// SIMATIC S7-200 project (STEP 7-Micro/WIN), CPU 224 REL 02.01

SYMBOL_TABLE USUARIO1
P_MARCHA         I0.0
P_PARO           I0.1
P_DESACTIVACION  I0.2
FCEL1            I0.3
FCEL2            I0.4
F_C_F_LINEA      I0.5
S_PRESION        I0.6
F_C_T2           I0.7
F_C_T3           I1.0
CT_M_1           Q0.0
CT_M_2           Q0.1
CT_M_3           Q0.2
P_DESPLA_P       Q0.3
P_ELEVACION      Q0.4
P_BAJADA         Q0.5
P_T3             Q0.6
MEM_CP           M10.1
MEM_CG           M10.3
PT_2             Q0.7
END_SYMBOL_TABLE

ORGANIZATION_BLOCK PRINCIPAL:OB1
TITLE=COMENTARIOS DEL PROGRAMA
BEGIN
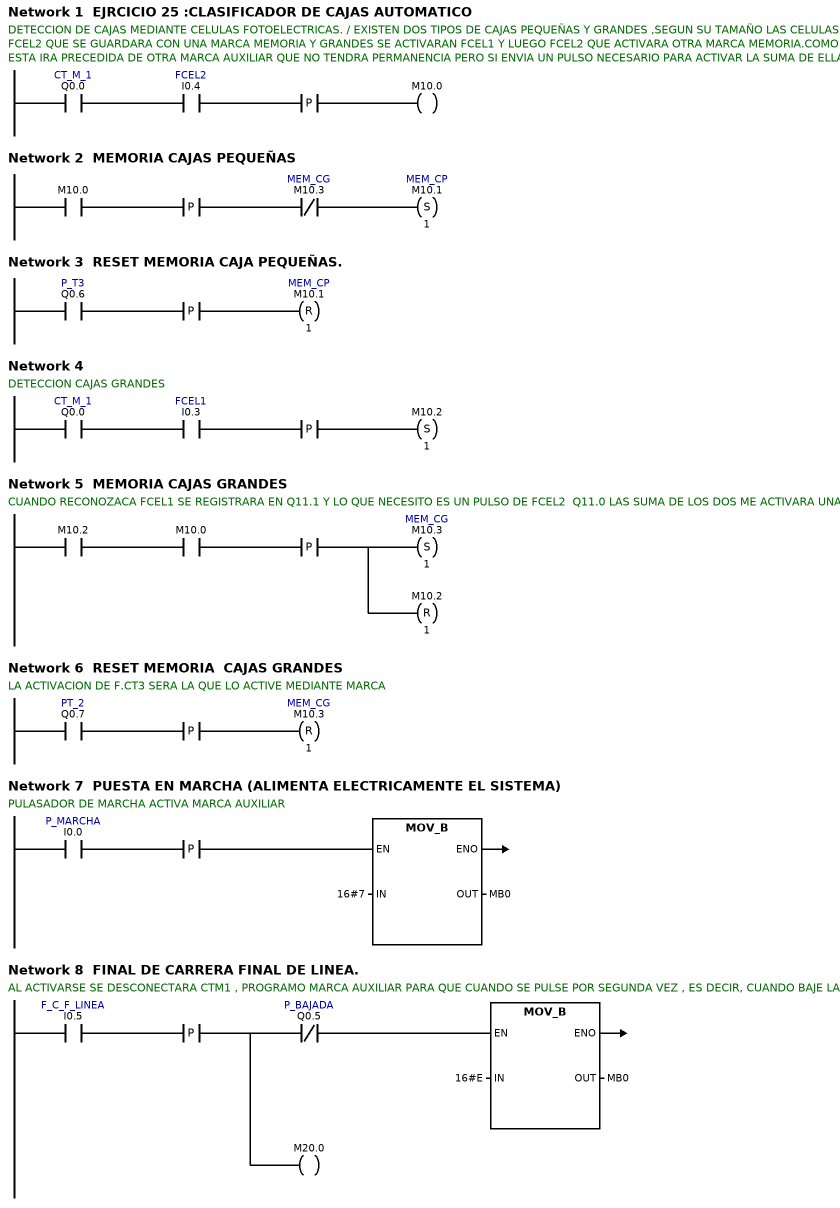
Network 1 // EJRCICIO 25 :CLASIFICADOR DE CAJAS AUTOMATICO
// DETECCION DE CAJAS MEDIANTE CELULAS FOTOELECTRICAS.
// EXISTEN DOS TIPOS DE CAJAS PEQUEÑAS Y GRANDES ,SEGUN SU TAMAÑO LAS CELULAS RECONOCERAN SI ES PEQUENA SOLO SE ACTIVA FCEL2 QUE SE GUARDARA CON UNA MARCA MEMORIA Y GRANDES SE ACTIVARAN FCEL1 Y LUEGO FCEL2 QUE ACTIVARA OTRA MARCA MEMORIA.COMO FCEL2 ES COMUN EN  LA PROGRAMACION DE ESTA IRA PRECEDIDA DE OTRA MARCA AUXILIAR QUE NO TENDRA PERMANENCIA PERO SI ENVIA UN PULSO NECESARIO PARA ACTIVAR LA SUMA DE ELLAS Y  CONTACTO CERRADO DELANTE DE MEMORIA FCEL2 EVITARA QUE SE ACTIVEN LAS DOS A LA VEZ.
// 
// 
// DETECCION CAJAS PEQUEÑAS
LD     CT_M_1:Q0.0
A      FCEL2:I0.4
EU
=      M10.0
Network 2 // MEMORIA CAJAS PEQUEÑAS 
LD     M10.0
EU
AN     MEM_CG:M10.3
S      MEM_CP:M10.1, 1
Network 3 // RESET MEMORIA CAJA PEQUEÑAS.
LD     P_T3:Q0.6
EU
R      MEM_CP:M10.1, 1
Network 4
// DETECCION CAJAS GRANDES
LD     CT_M_1:Q0.0
A      FCEL1:I0.3
EU
S      M10.2, 1
Network 5 // MEMORIA CAJAS GRANDES
// CUANDO RECONOZACA FCEL1 SE REGISTRARA EN Q11.1 Y LO QUE NECESITO ES UN PULSO DE FCEL2  Q11.0 LAS SUMA DE LOS DOS ME ACTIVARA UNA TERCERA QUE SERA LA DE MEMORIA Q11.3
LD     M10.2
A      M10.0
EU
S      MEM_CG:M10.3, 1
R      M10.2, 1
Network 6 // RESET MEMORIA  CAJAS GRANDES
// LA ACTIVACION DE F.CT3 SERA LA QUE LO ACTIVE MEDIANTE MARCA
LD     PT_2:Q0.7
EU
R      MEM_CG:M10.3, 1
Network 7 // PUESTA EN MARCHA (ALIMENTA ELECTRICAMENTE EL SISTEMA)
// PULASADOR DE MARCHA ACTIVA MARCA AUXILIAR 
LD     P_MARCHA:I0.0
EU
MOVB   16#7, MB0
Network 8 // FINAL DE CARRERA FINAL DE LINEA.
// AL ACTIVARSE SE DESCONECTARA CTM1 , PROGRAMO MARCA AUXILIAR PARA QUE CUANDO SE PULSE POR SEGUNDA VEZ , ES DECIR, CUANDO BAJE LA PLATAFORMA ACTIVE CTM1
LD     F_C_F_LINEA:I0.5
EU
LPS
AN     P_BAJADA:Q0.5
MOVB   16#E, MB0
LPP
=      M20.0
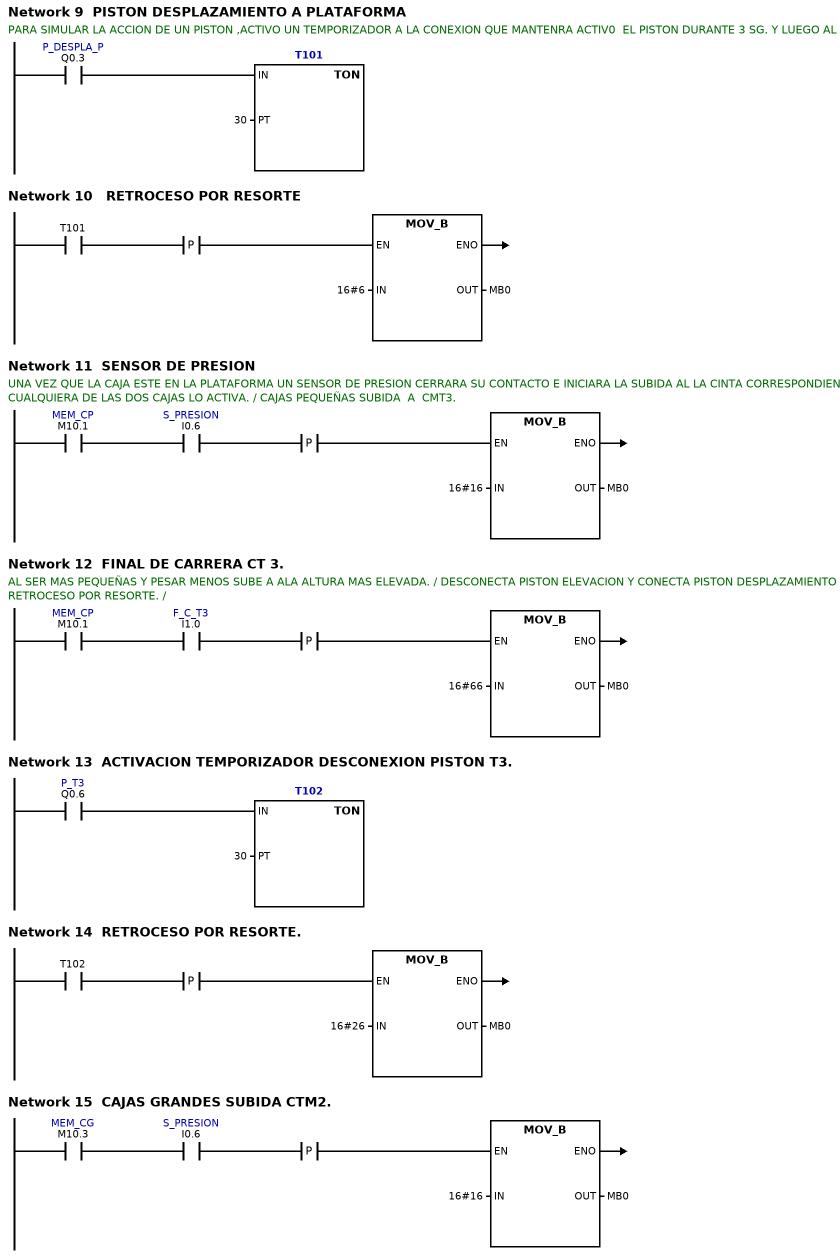
Network 9 // PISTON DESPLAZAMIENTO A PLATAFORMA
// PARA SIMULAR LA ACCION DE UN PISTON ,ACTIVO UN TEMPORIZADOR A LA CONEXION QUE MANTENRA ACTIV0  EL PISTON DURANTE 3 SG. Y LUEGO AL APAGARSE INICIA EL RETROCESO POR RESORTE.
LD     P_DESPLA_P:Q0.3
TON    T101, 30
Network 10 //  RETROCESO POR RESORTE
LD     T101
EU
MOVB   16#6, MB0
Network 11 // SENSOR DE PRESION 
// UNA VEZ QUE LA CAJA ESTE EN LA PLATAFORMA UN SENSOR DE PRESION CERRARA SU CONTACTO E INICIARA LA SUBIDA AL LA CINTA CORRESPONDIENTE . CALIBRADA DE TAL FORMA QUE EL PESO DE CUALQUIERA DE LAS DOS CAJAS LO ACTIVA.
// CAJAS PEQUEÑAS SUBIDA  A  CMT3.
LD     MEM_CP:M10.1
A      S_PRESION:I0.6
EU
MOVB   16#16, MB0
Network 12 // FINAL DE CARRERA CT 3.
// AL SER MAS PEQUEÑAS Y PESAR MENOS SUBE A ALA ALTURA MAS ELEVADA.
// DESCONECTA PISTON ELEVACION Y CONECTA PISTON DESPLAZAMIENTO A CTM 3 Y BAJADA REPOSO SIMULACION RETROCESO POR RESORTE.
// 
LD     MEM_CP:M10.1
A      F_C_T3:I1.0
EU
MOVB   16#66, MB0
Network 13 // ACTIVACION TEMPORIZADOR DESCONEXION PISTON T3. 
LD     P_T3:Q0.6
TON    T102, 30
Network 14 // RETROCESO POR RESORTE.
LD     T102
EU
MOVB   16#26, MB0
Network 15 // CAJAS GRANDES SUBIDA CTM2.
LD     MEM_CG:M10.3
A      S_PRESION:I0.6
EU
MOVB   16#16, MB0
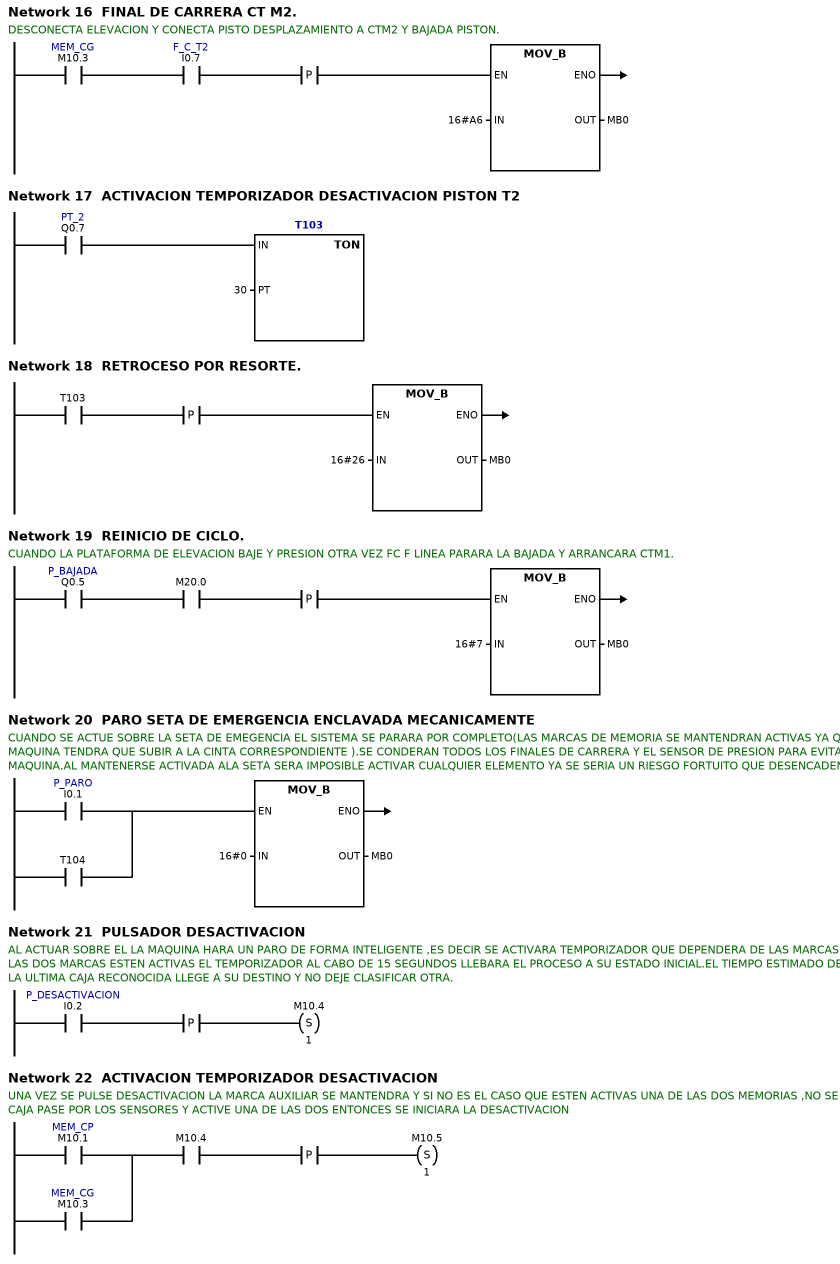
Network 16 // FINAL DE CARRERA CT M2.
// DESCONECTA ELEVACION Y CONECTA PISTO DESPLAZAMIENTO A CTM2 Y BAJADA PISTON.
LD     MEM_CG:M10.3
A      F_C_T2:I0.7
EU
MOVB   16#A6, MB0
Network 17 // ACTIVACION TEMPORIZADOR DESACTIVACION PISTON T2
LD     PT_2:Q0.7
TON    T103, 30
Network 18 // RETROCESO POR RESORTE.
LD     T103
EU
MOVB   16#26, MB0
Network 19 // REINICIO DE CICLO.
// CUANDO LA PLATAFORMA DE ELEVACION BAJE Y PRESION OTRA VEZ FC F LINEA PARARA LA BAJADA Y ARRANCARA CTM1.
LD     P_BAJADA:Q0.5
A      M20.0
EU
MOVB   16#7, MB0
Network 20 // PARO SETA DE EMERGENCIA ENCLAVADA MECANICAMENTE 
// CUANDO SE ACTUE SOBRE LA SETA DE EMEGENCIA EL SISTEMA SE PARARA POR COMPLETO(LAS MARCAS DE MEMORIA SE MANTENDRAN ACTIVAS YA QUE CUANDO SE REANUDE EL SISTEMA LA MAQUINA TENDRA QUE SUBIR A LA CINTA CORRESPONDIENTE ).SE CONDERAN TODOS LOS FINALES DE CARRERA Y EL SENSOR DE PRESION PARA EVITAR ACCIDENTEN MIENTRAS SE MANIPULE LA MAQUINA.AL MANTENERSE ACTIVADA ALA SETA SERA IMPOSIBLE ACTIVAR CUALQUIER ELEMENTO YA SE SERIA UN RIESGO FORTUITO QUE DESENCADENARIA UN ERROR FATAL.
LD     P_PARO:I0.1
O      T104
MOVB   16#0, MB0
Network 21 // PULSADOR DESACTIVACION
// AL ACTUAR SOBRE EL LA MAQUINA HARA UN PARO DE FORMA INTELIGENTE ,ES DECIR SE ACTIVARA TEMPORIZADOR QUE DEPENDERA DE LAS MARCAS DE MEMORIA , UNA VEZ SE PRESIONE Y UNA DE LAS DOS MARCAS ESTEN ACTIVAS EL TEMPORIZADOR AL CABO DE 15 SEGUNDOS LLEBARA EL PROCESO A SU ESTADO INICIAL.EL TIEMPO ESTIMADO DE DESCONEXION SERA EL OPORTUNO PARA QUE LA ULTIMA CAJA RECONOCIDA LLEGE A SU DESTINO Y NO DEJE CLASIFICAR OTRA.
LD     P_DESACTIVACION:I0.2
EU
S      M10.4, 1
Network 22 // ACTIVACION TEMPORIZADOR DESACTIVACION
// UNA VEZ SE PULSE DESACTIVACION LA MARCA AUXILIAR SE MANTENDRA Y SI NO ES EL CASO QUE ESTEN ACTIVAS UNA DE LAS DOS MEMORIAS ,NO SE ACTIVARA EL TEMPORIZADOR HASTA QUE LA CAJA PASE POR LOS SENSORES Y ACTIVE UNA DE LAS DOS ENTONCES SE INICIARA LA DESACTIVACION
LD     MEM_CP:M10.1
O      MEM_CG:M10.3
A      M10.4
EU
S      M10.5, 1
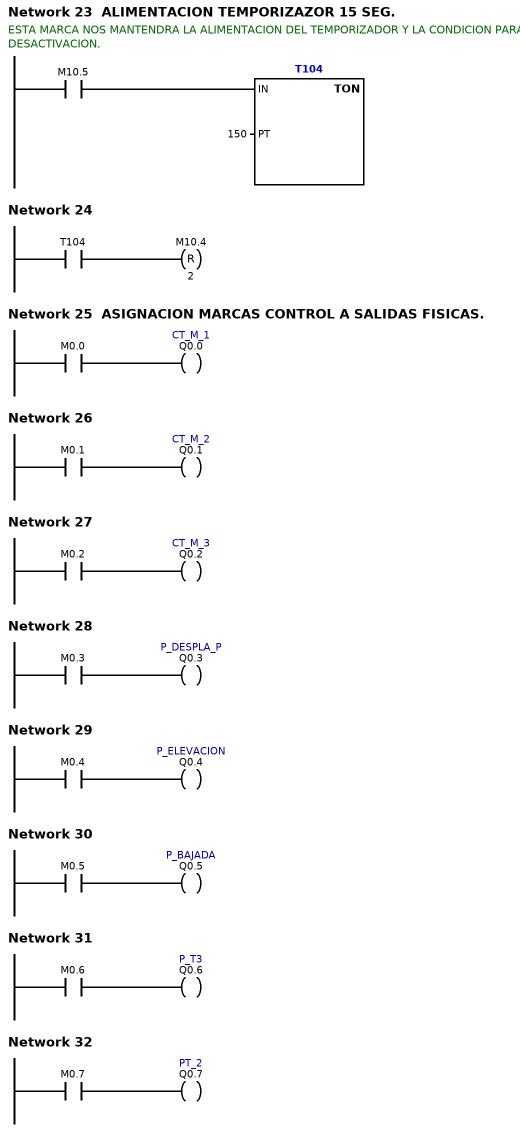
Network 23 // ALIMENTACION TEMPORIZAZOR 15 SEG.
// ESTA MARCA NOS MANTENDRA LA ALIMENTACION DEL TEMPORIZADOR Y LA CONDICION PARA QUE ESTE ALIMENTADA ES QUE ESTE UNA DE LAS DOS MEMORIAS ACTIVAS Y SE HALLA PULSADO DESACTIVACION.
LD     M10.5
TON    T104, 150
Network 24
LD     T104
R      M10.4, 2
Network 25 // ASIGNACION MARCAS CONTROL A SALIDAS FISICAS.
LD     M0.0
=      CT_M_1:Q0.0
Network 26
LD     M0.1
=      CT_M_2:Q0.1
Network 27
LD     M0.2
=      CT_M_3:Q0.2
Network 28
LD     M0.3
=      P_DESPLA_P:Q0.3
Network 29
LD     M0.4
=      P_ELEVACION:Q0.4
Network 30
LD     M0.5
=      P_BAJADA:Q0.5
Network 31
LD     M0.6
=      P_T3:Q0.6
Network 32
LD     M0.7
=      PT_2:Q0.7
END_ORGANIZATION_BLOCK
